// SIMATIC S7-200 project (STEP 7-Micro/WIN), CPU 221 REL 01.10

ORGANIZATION_BLOCK PRINCIPAL:OB1
TITLE=PRÁCTICA 11 Grafcet B - JEVG
BEGIN
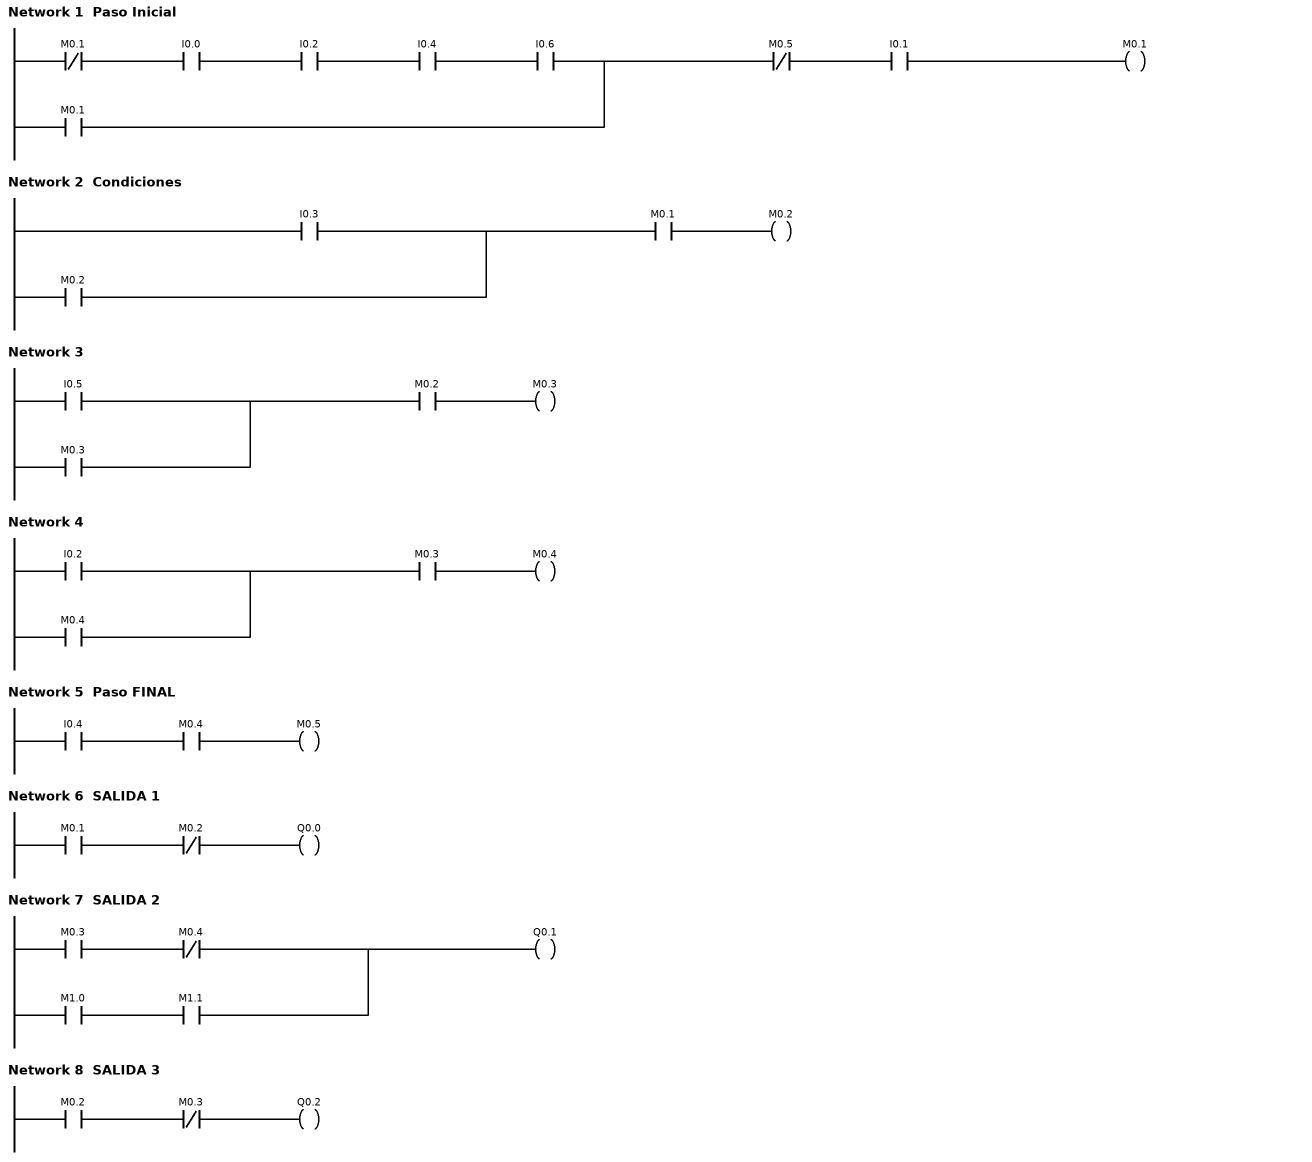
Network 1 // Paso Inicial
// (network saved uncompiled; LAD cells follow)
// row 0: c0 -|/|- M0.1  c1 -| |- I0.0  c2 -| |- I0.2  c3 -| |- I0.4  c4 -| |- I0.6 v  c5 --  c6 -|/|- M0.5  c7 -| |- I0.1  c8 --  c9 -( ) M0.1
// row 1: c0 -| |- M0.1  c1 --  c2 --  c3 --  c4 -- ^
Network 2 // Condiciones
// (network saved uncompiled; LAD cells follow)
// row 0: c0 --  c1 --  c2 -| |- I0.3  c3 -- v  c4 --  c5 -| |- M0.1  c6 -( ) M0.2
// row 1: c0 -| |- M0.2  c1 --  c2 --  c3 -- ^
Network 3
// (network saved uncompiled; LAD cells follow)
// row 0: c0 -| |- I0.5  c1 -- v  c2 --  c3 -| |- M0.2  c4 -( ) M0.3
// row 1: c0 -| |- M0.3  c1 -- ^
Network 4
// (network saved uncompiled; LAD cells follow)
// row 0: c0 -| |- I0.2  c1 -- v  c2 --  c3 -| |- M0.3  c4 -( ) M0.4
// row 1: c0 -| |- M0.4  c1 -- ^
Network 5 // Paso FINAL
LD     I0.4
A      M0.4
=      M0.5
Network 6 // SALIDA 1
// (network saved uncompiled; LAD cells follow)
// row 0: c0 -| |- M0.1  c1 -|/|- M0.2  c2 -( ) Q0.0
Network 7 // SALIDA 2
// (network saved uncompiled; LAD cells follow)
// row 0: c0 -| |- M0.3  c1 -|/|- M0.4  c2 -- v  c3 --  c4 -( ) Q0.1
// row 1: c0 -| |- M1.0  c1 -| |- M1.1  c2 -- ^
Network 8 // SALIDA 3
// (network saved uncompiled; LAD cells follow)
// row 0: c0 -| |- M0.2  c1 -|/|- M0.3  c2 -( ) Q0.2
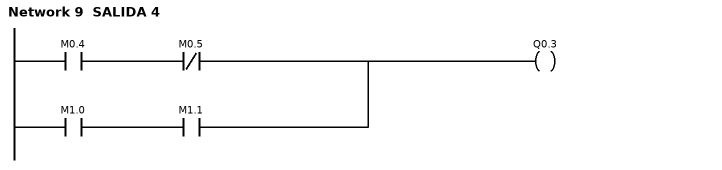
Network 9 // SALIDA 4
// (network saved uncompiled; LAD cells follow)
// row 0: c0 -| |- M0.4  c1 -|/|- M0.5  c2 -- v  c3 --  c4 -( ) Q0.3
// row 1: c0 -| |- M1.0  c1 -| |- M1.1  c2 -- ^
END_ORGANIZATION_BLOCK
